Staubli VAL3: remErrPower.pgx

program remErrPower(string& sReturn[] (dimensions=1))
begin
  // Error raised when we try to move the robot
  // but the arm is not powered
  //
  logMsg("call remErrPower")
  sReturn="ERROR 202"
  sReturn=sReturn+": Arm is not powered."
  putln(sReturn)
  logMsg(sReturn)
end
